TYPE ST_FeedbackLeica :
STRUCT
	pos: ARRAY[0..2] OF LREAL;
	quat: ARRAY[0..3] OF LREAL;
END_STRUCT
END_TYPE

(* stored: Version 1.1.0.1, ProductVersion 3.1.4022.7
   DUT ST_FeedbackLeica: Id {27e2f734-a908-46c7-b4c1-0957dce28692} *)
